ABB RobotStudio station: mysolution1_1_20200829-160056.rsstn

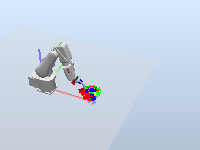
Station mysolution1 (saved by RobotStudio 20.1.9014.1)
Controller Controller1, task T_ROB1: task frame (RAPID world) sits at (50, 0, 0) mm in the station
Controller Controller1
  mechanical unit ROB_1: IRB120_3_58__01, 6 joints, base frame (0, 0, 0) mm
Layout (positions relative to the parent item):
  - IRB120_3_58__01 [mechanism, from Robots\IRB120_3_58_G_01.rslib] at (50, 0, 0) mm; joint values [0.1009, 0.5466, 0.7336, -0.3396, -0.5635, -0.103] (rad or m)
  - AssemblyWeldingTorch [part] at (321.3, 37.78, 165.01) mm, rotated rx -42.5 ry -9.85 rz -61.52 deg
  - Workpiece_2 [part] at (580, 20, 8) mm, rotated rx 90 ry 0 rz 90 deg
Attachment: AssemblyWeldingTorch is attached to IRB120_3_58__01 / Link6
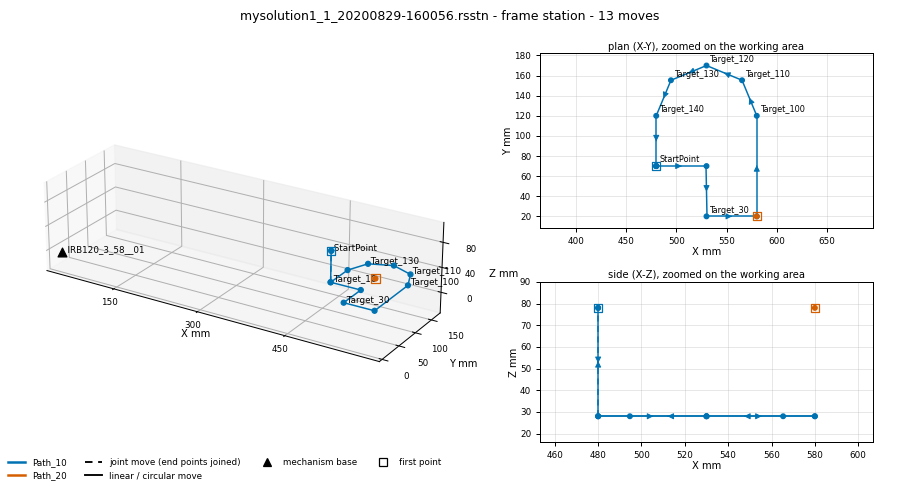
[picture p0: tool path of mysolution1_1_20200829-160056.rsstn in frame station, 13 of 13 moves have a stored position in this frame; points joined in program order, loops and branches not executed]
Targets, tools, work objects and paths stored in the station, written as RAPID:
! task T_ROB1
MODULE CalibData
  TASK PERS tooldata WeldingTorch:=[TRUE,[[35,0,150.231],[0.965925826,0,0.258819045,0]],[1,[0,0,1],[1,0,0,0],0,0,0]];
  TASK PERS wobjdata Workobject_2:=[FALSE,TRUE,"",[[530,20,8],[0.707106781,0,0,0.707106782]],[[0,0,0],[1,0,0,0]]];
ENDMODULE

! task T_ROB1
MODULE Module1
  CONST robtarget LiftOffPoint:=[[0,0,70],[0.086824089,0.492403876,0.852868532,-0.150383733],[-1,1,2,0],[9E+09,9E+09,9E+09,9E+09,9E+09,9E+09]];
  CONST robtarget Target_10:=[[50,100,20],[0.086824089,0.492403876,0.852868532,-0.150383733],[0,-1,-1,1],[9E+09,9E+09,9E+09,9E+09,9E+09,9E+09]];
  CONST robtarget Target_20:=[[50,50,20],[0.086824089,0.492403876,0.852868532,-0.150383733],[0,-1,-1,1],[9E+09,9E+09,9E+09,9E+09,9E+09,9E+09]];
  CONST robtarget Target_30:=[[0,50,20],[0.086824089,0.492403876,0.852868532,-0.150383733],[-1,-1,-1,1],[9E+09,9E+09,9E+09,9E+09,9E+09,9E+09]];
  CONST robtarget Target_40:=[[0,0,20],[0.086824089,0.492403876,0.852868532,-0.150383733],[-1,-1,0,1],[9E+09,9E+09,9E+09,9E+09,9E+09,9E+09]];
  CONST robtarget StartPoint:=[[50,100,70],[0.086824089,0.492403876,0.852868532,-0.150383733],[0,-1,-1,1],[9E+09,9E+09,9E+09,9E+09,9E+09,9E+09]];
  CONST robtarget Target_50:=[[100,0,20],[0.707106781,-0.707106781,0,0],[0,0,0,0],[9E+09,9E+09,9E+09,9E+09,9E+09,9E+09]];
  CONST robtarget Target_60:=[[135.355339059,14.644660941,20],[0.653281482,-0.653281482,-0.27059805,0.27059805],[0,0,0,0],[9E+09,9E+09,9E+09,9E+09,9E+09,9E+09]];
  CONST robtarget Target_70:=[[150,50,20],[0.5,-0.5,-0.5,0.5],[0,0,0,0],[9E+09,9E+09,9E+09,9E+09,9E+09,9E+09]];
  CONST robtarget Target_80:=[[135.355318525,85.355308775,19.99996882],[0.27059809,-0.270598108,-0.653281464,0.65328146],[-1,0,0,0],[9E+09,9E+09,9E+09,9E+09,9E+09,9E+09]];
  CONST robtarget Target_90:=[[100,100,20],[0,0,-0.707106781,0.707106781],[0,0,0,0],[9E+09,9E+09,9E+09,9E+09,9E+09,9E+09]];
  CONST robtarget Target_10_2:=[[50,100,20],[0.086824089,0.492403876,0.852868532,-0.150383733],[-1,-1,-1,1],[9E+09,9E+09,9E+09,9E+09,9E+09,9E+09]];
  CONST robtarget StartPoint_2:=[[50,100,70],[0.086824089,0.492403876,0.852868532,-0.150383733],[0,-1,-1,1],[9E+09,9E+09,9E+09,9E+09,9E+09,9E+09]];
  CONST robtarget Target_100:=[[100,-0.000000141,20],[0,1,-0.000000001,0],[0,1,-1,1],[9E+09,9E+09,9E+09,9E+09,9E+09,9E+09]];
  CONST robtarget Target_110:=[[135.35533908,14.64466075,20],[0,0.923879533,0.382683432,0],[0,1,-1,1],[9E+09,9E+09,9E+09,9E+09,9E+09,9E+09]];
  CONST robtarget Target_120:=[[150.000000071,49.999999788,20],[0,0.707106782,0.707106781,0],[0,1,-2,1],[9E+09,9E+09,9E+09,9E+09,9E+09,9E+09]];
  CONST robtarget Target_130:=[[135.35533918,85.355338868,20],[0,0.382683434,0.923879532,0],[0,-2,0,1],[9E+09,9E+09,9E+09,9E+09,9E+09,9E+09]];
  CONST robtarget Target_140:=[[100.000000141,99.999999859,20],[0,0.000000001,1,0],[0,-2,0,1],[9E+09,9E+09,9E+09,9E+09,9E+09,9E+09]];
  CONST robtarget Target_10_3:=[[50,100,20],[0.086824089,0.492403876,0.852868532,-0.150383733],[0,-1,-1,1],[9E+09,9E+09,9E+09,9E+09,9E+09,9E+09]];
  CONST robtarget StartPoint_3:=[[50,100,70],[0.086824089,0.492403876,0.852868532,-0.150383733],[0,-1,-1,1],[9E+09,9E+09,9E+09,9E+09,9E+09,9E+09]];
  PROC Path_10()
    MoveJ StartPoint,v1000,z100,WeldingTorch\WObj:=Workobject_2;
    MoveL Target_10,v1000,z100,WeldingTorch\WObj:=Workobject_2;
    MoveL Target_20,v1000,z100,WeldingTorch\WObj:=Workobject_2;
    MoveL Target_30,v1000,z100,WeldingTorch\WObj:=Workobject_2;
    MoveL Target_40,v1000,z100,WeldingTorch\WObj:=Workobject_2;
    MoveL Target_100,v100,z10,WeldingTorch\WObj:=Workobject_2;
    MoveL Target_110,v100,z10,WeldingTorch\WObj:=Workobject_2;
    MoveL Target_120,v100,z10,WeldingTorch\WObj:=Workobject_2;
    MoveL Target_130,v100,z10,WeldingTorch\WObj:=Workobject_2;
    MoveL Target_140,v100,z10,WeldingTorch\WObj:=Workobject_2;
    MoveL Target_10_3,v1000,z100,WeldingTorch\WObj:=Workobject_2;
    MoveJ StartPoint_3,v1000,z100,WeldingTorch\WObj:=Workobject_2;
  ENDPROC
  PROC Main()
    Path_10;
  ENDPROC
  PROC Path_20()
    MoveJ LiftOffPoint,v1000,z100,WeldingTorch\WObj:=Workobject_2;
  ENDPROC
ENDMODULE

